# EPICS autosave request: iocBoot/iocdmm7510/auto_settings_dmm7510.req
file "dmm7510_settings.req",                P=$(P),  R=$(R)
